TYPE ST_OutputsFunctionForks :
STRUCT
	ForkStatus					: ST_ForkState;//out to element
END_STRUCT
END_TYPE

(* stored: Version 1.1.0.1, ProductVersion 3.1.4024.9
   DUT ST_OutputsFunctionForks: Id {27b7b2f1-15ea-4132-8462-2dd084805aa9} *)
